FUNCTION_BLOCK FB_EstacionRestaurar_SFC
VAR_INPUT
    // SFC-Flags
    SFCPause: BOOL;
    SFCReset: BOOL;
    
    // Indicadores de sincronizacion
    Ack: BOOL := TRUE;
    Execute: BOOL;
    
    // Entradas
    ManipuladorDetras: BOOL; // Sobre el pale
    ManipuladorMedio: BOOL := TRUE; // En la vertical
    PrensadorArriba: BOOL := TRUE;
END_VAR
VAR_OUTPUT
    // Indicadores de sincronizacion
    Done: BOOL;
    Ready: BOOL;
    
    // Salidas
    ManipuladorAdelante: BOOL; // Hacia el punto de trasvase de la prensa
    ManipuladorAtras: BOOL; // Hacia el pale
    PrensadorSube: BOOL;    
END_VAR
VAR
END_VAR

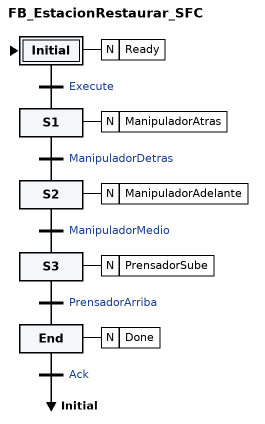
INITIAL_STEP Initial:
    Ready(N);
END_STEP
TRANSITION FROM Initial TO S1
    := Execute;
END_TRANSITION
STEP S1:
    ManipuladorAtras(N);
END_STEP
TRANSITION FROM S1 TO S2
    := ManipuladorDetras;
END_TRANSITION
STEP S2:
    ManipuladorAdelante(N);
END_STEP
TRANSITION FROM S2 TO S3
    := ManipuladorMedio;
END_TRANSITION
STEP S3:
    PrensadorSube(N);
END_STEP
TRANSITION FROM S3 TO End
    := PrensadorArriba;
END_TRANSITION
STEP End:
    Done(N);
END_STEP
TRANSITION FROM End TO Initial
    := Ack;
END_TRANSITION

END_FUNCTION_BLOCK

(* stored: Version 1.1.0.1, ProductVersion 3.1.4024.12
   POU FB_EstacionRestaurar_SFC: Id {e735efd1-7aba-4b5c-bc7a-4a8e4ddd46db}, SpecialFunc None *)
